# EPICS substitutions: ek9000App/Db/EL9505_mbbiDirect.substitutions
file EL9505.template
{       pattern
        {
                TERMINAL,

        }
        {
        }
}
